{attribute 'GeneratedUsingTerminal: EL3201-0030-0022'}
{attribute addProperty BoxType "EL3201-0030-0022"}
{attribute addProperty Description "EL3201-0030 1Ch. Ana. Input PT100 (RTD), High Precision, external calibrated"}
{attribute addProperty Physics "KK"}
{attribute addProperty Id "RTDAT %I*AI_Standard_Channel_4A3944819WcStateAT %I*WcState_9091E0EB2InfoDataAT %I*InfoData_32EB74EA10"}
{attribute addProperty CRC "4084989573"}
{attribute addProperty Size "21"}
TYPE EL3201_F37BFE85 EXTENDS EtcSlaveTerminalBase_947E5A46 :
STRUCT
	{attribute addProperty Name "RTD"}
	RTD : AI_Standard_Channel_4A394481;
	{attribute addProperty Name "WcState"}
	WcState : WcState_9091E0EB;
	{attribute addProperty Name "InfoData"}
	InfoData : InfoData_32EB74EA;
END_STRUCT
END_TYPE

(* stored: Version 1.2.0.0, ProductVersion 3.1.4024.11
   DUT EL3201_F37BFE85: Id {373f6657-5a33-4ca2-b3a6-7bb252e9550e} *)
